(* PLC project lng-production, Generated TextualNotationConverter 1.0 *)
(* stored: creationDateTime 2025-07-30T12:00:00, modificationDateTime 2025-09-16T14:04:18 *)

FUNCTION_BLOCK ANALOG_IN
  VAR_INPUT
    Name : STRING;
    Description : STRING;
    Raw_Signal : REAL;
    PV_High : REAL;
    PV_Low : REAL;
    Scaling_Slope : REAL;
    Scaling_Offset : REAL;
    Alarm_Enable : BOOL;
  END_VAR
  VAR_OUTPUT
    PV : REAL;
    High_Alarm : BOOL;
    Low_Alarm : BOOL;
    General_Fault : BOOL;
  END_VAR

            
          
END_FUNCTION_BLOCK

FUNCTION_BLOCK RATIO_CONTROL
  VAR_INPUT
    Name : STRING;
    Description : STRING;
    Auto : BOOL;
    PrimaryPV : REAL;
    SecondaryPV : REAL;
    RatioSP : REAL;
    Bias : REAL;
    TrimKp : REAL;
    TrimTi : STRING;
    MV_MIN : REAL;
    MV_MAX : REAL;
    ManOut : REAL;
    Inhibit : BOOL;
  END_VAR
  VAR_OUTPUT
    SlaveSP : REAL;
    ActiveRatio : REAL;
    RatioErr : REAL;
  END_VAR

            
          
END_FUNCTION_BLOCK

FUNCTION_BLOCK VALVE_ELECTRIC
  VAR_INPUT
    Name : STRING;
    Description : STRING;
    Control_Signal : REAL;
    Manual_Mode : BOOL;
    Manual_Position : REAL;
    Open_Limit : REAL;
    Close_Limit : REAL;
    Timeout : STRING;
    Inhibit : BOOL;
  END_VAR
  VAR_OUTPUT
    Valve_Position : REAL;
    Feedback_Pos : REAL;
    Valve_Moving : BOOL;
    Position_Error : BOOL;
    Alarm : BOOL;
  END_VAR

            
          
END_FUNCTION_BLOCK

PROGRAM Section2
  VAR
    FT_101_Flow_PV : REAL;
    IT_102_Flow_PV : REAL;
    DP_101_DiffP_PV : REAL;
    DP_102_DiffP_PV : REAL;
    LT_101_Level_PV : REAL;
    IIC_101_LiqSepFlow_SP : REAL;
  END_VAR
  VAR
    DP-101 : ANALOG_IN;
    DP-102 : ANALOG_IN;
    FT-101 : ANALOG_IN;
    IT-102 : ANALOG_IN;
    LT-101 : ANALOG_IN;
    IIC-101 : RATIO_CONTROL;
    LCV-101 : VALVE_ELECTRIC;
  END_VAR

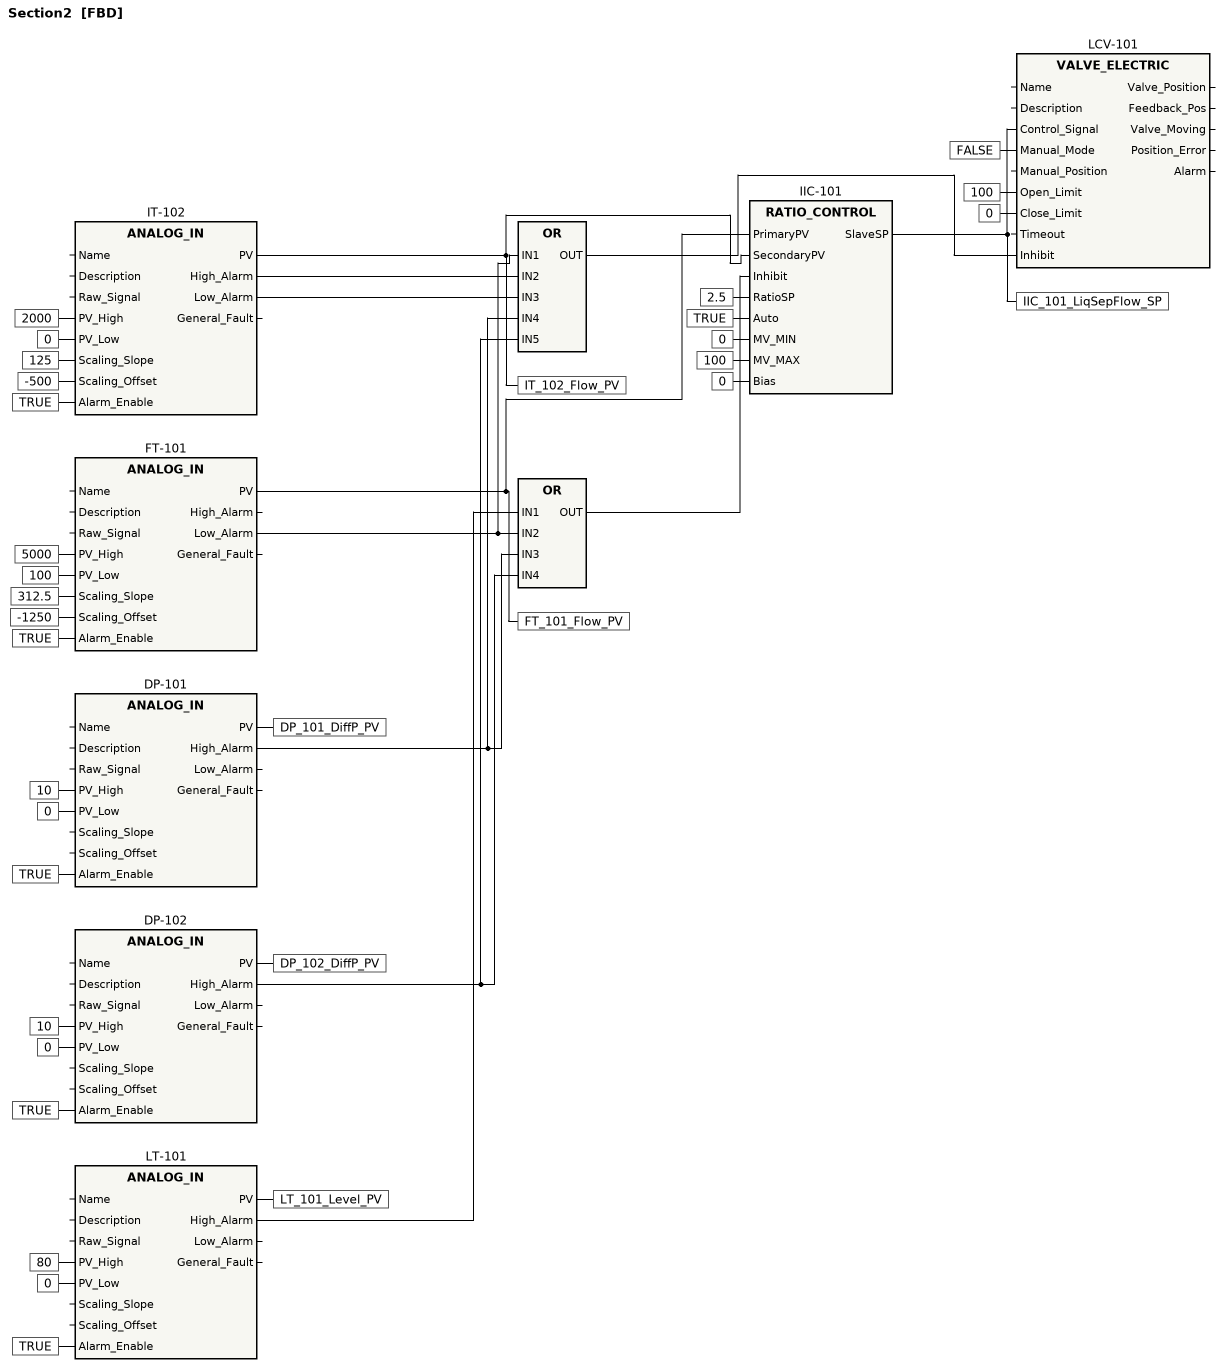
(* FBD diagram, written out as Structured Text *)
DP-101(PV_High := 10, PV_Low := 0, Alarm_Enable := TRUE);
DP_101_DiffP_PV := DP-101.PV;
DP-102(PV_High := 10, PV_Low := 0, Alarm_Enable := TRUE);
DP_102_DiffP_PV := DP-102.PV;
FT-101(PV_High := 5000, PV_Low := 100, Scaling_Slope := 312.5, Scaling_Offset := -1250, Alarm_Enable := TRUE);
FT_101_Flow_PV := FT-101.PV;
IT-102(PV_High := 2000, PV_Low := 0, Scaling_Slope := 125, Scaling_Offset := -500, Alarm_Enable := TRUE);
LT-101(PV_High := 80, PV_Low := 0, Alarm_Enable := TRUE);
IIC-101(PrimaryPV := FT-101.PV, SecondaryPV := IT-102.PV, Inhibit := LT-101.High_Alarm OR FT-101.Low_Alarm OR DP-101.High_Alarm OR DP-102.High_Alarm, RatioSP := 2.5, Auto := TRUE, MV_MIN := 0, MV_MAX := 100, Bias := 0);
IIC_101_LiqSepFlow_SP := IIC-101.SlaveSP;
IT_102_Flow_PV := IT-102.PV;
LT_101_Level_PV := LT-101.PV;
LCV-101(Control_Signal := IIC-101.SlaveSP, Manual_Mode := FALSE, Open_Limit := 100, Close_Limit := 0, Inhibit := FT-101.Low_Alarm OR IT-102.High_Alarm OR IT-102.Low_Alarm OR DP-101.High_Alarm OR DP-102.High_Alarm);
END_PROGRAM

FUNCTION_BLOCK BOOL_IN
  VAR_INPUT
    Name : STRING;
    Description : STRING;
    Bool_In : BOOL;
    Alarm_OnTrue : BOOL;
    Alarm_OnFalse : BOOL;
    Latch_Enable : BOOL;
    Reset_Latch : BOOL;
  END_VAR
  VAR_OUTPUT
    Bool_Out : BOOL;
    Alarm_Active : BOOL;
    Latched_Status : BOOL;
  END_VAR

            
          
END_FUNCTION_BLOCK

FUNCTION_BLOCK DIGITAL_IN
  VAR_INPUT
    Name : STRING;
    Description : STRING;
    DI_Raw : BOOL;
    DebounceTime : STRING;
    EnableAlarm : BOOL;
  END_VAR
  VAR_OUTPUT
    DI_Out : BOOL;
    Fault_State : BOOL;
  END_VAR

            
          
END_FUNCTION_BLOCK

FUNCTION_BLOCK DUTY_STANDBY
  VAR_INPUT
    Name : STRING;
    Description : STRING;
    Enable : BOOL;
    StartRequest : BOOL;
    AlternateEnable : BOOL;
    ForcePumpA : BOOL;
    ForcePumpB : BOOL;
    DutyElapsed : BOOL;
    MinRunElapsed : BOOL;
    SwitchoverDelayElapsed : BOOL;
    StartTimeoutElapsed : BOOL;
    PumpA_RunFB : BOOL;
    PumpB_RunFB : BOOL;
    PumpA_Fault : BOOL;
    PumpB_Fault : BOOL;
    Reset : BOOL;
    Inhibit : BOOL;
  END_VAR
  VAR_OUTPUT
    CmdPumpA : BOOL;
    CmdPumpB : BOOL;
    ActiveIsA : BOOL;
    SwitchedDueToDuty : BOOL;
    SwitchedDueToFailure : BOOL;
    Alarm_FailedStart_A : BOOL;
    Alarm_FailedStart_B : BOOL;
    Alarm_NoAvailablePump : BOOL;
  END_VAR

            
          
END_FUNCTION_BLOCK

FUNCTION_BLOCK MOTOR_2SPD
  VAR_INPUT
    Name : STRING;
    Description : STRING;
    Start_Cmd : BOOL;
    Stop_Cmd : BOOL;
    Speed_High_Cmd : BOOL;
    Speed_Low_Cmd : BOOL;
    Inhibit : BOOL;
  END_VAR
  VAR_OUTPUT
    Motor_Start_Out : BOOL;
    FB_Running : BOOL;
    FB_Trip : BOOL;
    FB_HighSpeed : BOOL;
    FB_LowSpeed : BOOL;
    Alarm_Speed_Error : BOOL;
  END_VAR

            
          
END_FUNCTION_BLOCK

FUNCTION_BLOCK MOTOR_ON_OFF
  VAR_INPUT
    Name : STRING;
    Description : STRING;
    Start_Cmd : BOOL;
    Stop_Cmd : BOOL;
    Start_Delay : STRING;
    MinRunTime : STRING;
    Inhibit : BOOL;
  END_VAR
  VAR_OUTPUT
    Motor_Start_Out : BOOL;
    FB_Running : BOOL;
    FB_Trip : BOOL;
    Alarm_Start_Fail : BOOL;
    Alarm_Stop_Fail : BOOL;
  END_VAR

            
          
END_FUNCTION_BLOCK

FUNCTION_BLOCK MOTOR_VSD
  VAR_INPUT
    Name : STRING;
    Description : STRING;
    Start_Cmd : BOOL;
    Stop_Cmd : BOOL;
    Speed_SP : REAL;
    Accel_Ramp : STRING;
    Decel_Ramp : STRING;
    Inhibit : BOOL;
  END_VAR
  VAR_OUTPUT
    Speed_Out : REAL;
    FB_Running : BOOL;
    FB_Fault : BOOL;
    FB_Ready : BOOL;
    FB_ActualSpeed : REAL;
    Alarm_Speed_Deviation : BOOL;
    Alarm_Comm_Fail : BOOL;
  END_VAR

            
          
END_FUNCTION_BLOCK

FUNCTION_BLOCK PID_BASIC
  VAR_INPUT
    Name : STRING;
    Description : STRING;
    AUTO : BOOL;
    PV : REAL;
    SP : REAL;
    MV_MIN : REAL;
    MV_MAX : REAL;
    X0 : REAL;
    KP : REAL;
    TR : REAL;
    TD : REAL;
    PV_High : REAL;
    PV_Low : REAL;
    Deviation_Limit : REAL;
    Inhibit : BOOL;
  END_VAR
  VAR_OUTPUT
    PV_High_Alarm : BOOL;
    PV_Low_Alarm : BOOL;
    Deviation_Alarm : BOOL;
    XOUT : REAL;
  END_VAR

            
          
END_FUNCTION_BLOCK

FUNCTION_BLOCK SPLIT_RANGE
  VAR_INPUT
    Name : STRING;
    Description : STRING;
    IN : REAL;
    Split_Point : REAL;
    Output1_Start : REAL;
    Output1_End : REAL;
    Output2_Start : REAL;
    Output2_End : REAL;
  END_VAR
  VAR_OUTPUT
    OUT1 : REAL;
    OUT2 : REAL;
  END_VAR

            
          
END_FUNCTION_BLOCK

FUNCTION_BLOCK VALVE_ON_OFF
  VAR_INPUT
    Name : STRING;
    Description : STRING;
    Open_Cmd : BOOL;
    Close_Cmd : BOOL;
    Timeout : STRING;
    Inhibit : BOOL;
  END_VAR
  VAR_OUTPUT
    FB_Opened : BOOL;
    FB_Closed : BOOL;
    Valve_Open_Out : BOOL;
    Valve_Close_Out : BOOL;
    Alarm_Position_Error : BOOL;
    Alarm_General : BOOL;
  END_VAR

            
          
END_FUNCTION_BLOCK

FUNCTION_BLOCK VOTING_ANALOG
  VAR_INPUT
    Name : STRING;
    Description : STRING;
    Input1 : REAL;
    Input2 : REAL;
    Input3 : REAL;
    Deviation_Limit : REAL;
    Voting_Scheme : STRING;
    EnableAlarm : BOOL;
    Inhibit : BOOL;
  END_VAR
  VAR_OUTPUT
    Voted_Output : REAL;
    Sensor1_Fault : BOOL;
    Sensor2_Fault : BOOL;
    Sensor3_Fault : BOOL;
    Alarm_Voting_Error : BOOL;
    Healthy_Sensors_Count : INT;
  END_VAR

            
          
END_FUNCTION_BLOCK

PROGRAM Section3
  VAR
    TT201_Temperature_PV : REAL;
    PT201_FlashTankPressure_PV : REAL;
    LT201_AbsorberLevel_PV : REAL;
    AI201_CO2_PV : REAL;
    TIC201_MV_SteamValveCmd : REAL;
  END_VAR
  VAR
    AI-201 : ANALOG_IN;
    LT-201 : ANALOG_IN;
    PT-201 : ANALOG_IN;
    TT-201 : ANALOG_IN;
    TIC-201 : PID_BASIC;
    FV-101 : VALVE_ELECTRIC;
  END_VAR
  VAR  (* added by the conversion: wires and edge detectors of the diagram *)
    _OR43_OUT : BOOL;
  END_VAR

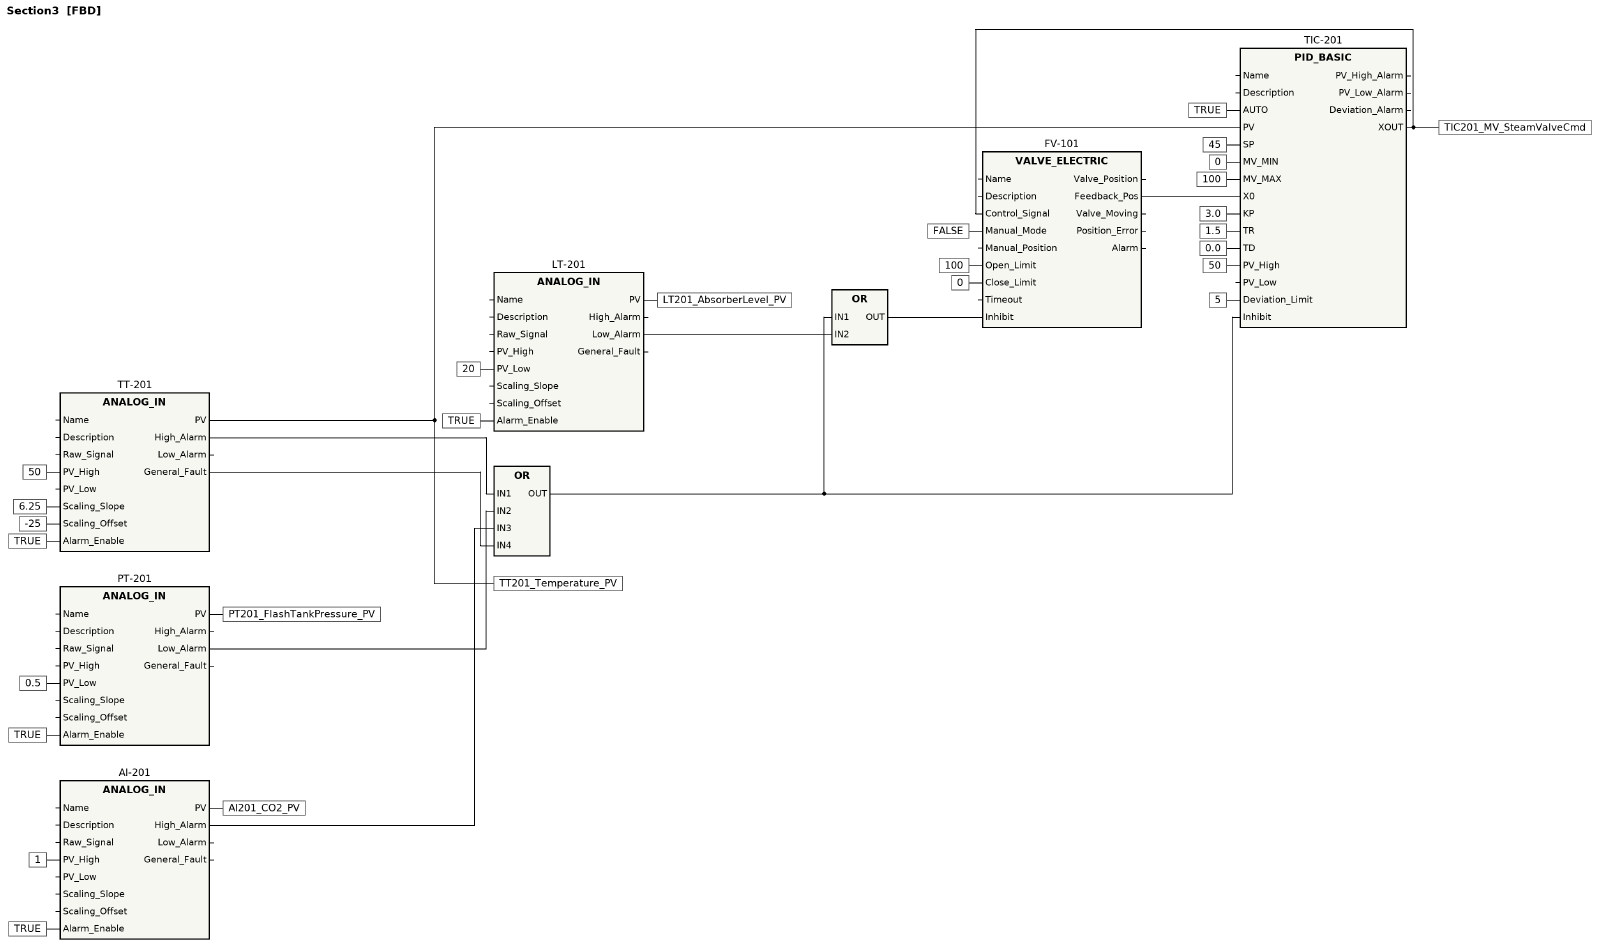
(* FBD diagram, written out as Structured Text *)
AI-201(PV_High := 1, Alarm_Enable := TRUE);
AI201_CO2_PV := AI-201.PV;
LT-201(PV_Low := 20, Alarm_Enable := TRUE);
LT201_AbsorberLevel_PV := LT-201.PV;
PT-201(PV_Low := 0.5, Alarm_Enable := TRUE);
PT201_FlashTankPressure_PV := PT-201.PV;
TT-201(PV_High := 50, Scaling_Slope := 6.25, Scaling_Offset := -25, Alarm_Enable := TRUE);
_OR43_OUT := TT-201.High_Alarm OR PT-201.Low_Alarm OR AI-201.High_Alarm OR TT-201.General_Fault;
FV-101(Control_Signal := TIC-201.XOUT, Manual_Mode := FALSE, Open_Limit := 100, Close_Limit := 0, Inhibit := _OR43_OUT OR LT-201.Low_Alarm);
TIC-201(AUTO := TRUE, PV := TT-201.PV, SP := 45, MV_MIN := 0, MV_MAX := 100, X0 := FV-101.Feedback_Pos, KP := 3.0, TR := 1.5, TD := 0.0, PV_High := 50, Deviation_Limit := 5, Inhibit := _OR43_OUT);
TIC201_MV_SteamValveCmd := TIC-201.XOUT;
TT201_Temperature_PV := TT-201.PV;
END_PROGRAM

PROGRAM Section4
  VAR
    AI302_H2O_Outlet_PV : REAL;
    AI303_Hg_Permissive_PV : REAL;
    AI304_H2O_RatioOpt_PV : REAL;
    FT301_FeedGasFlow_PV : REAL;
    DP301_MolSieveBed_DP_PV : REAL;
    FFIC303_RegenFlow_SP_to_FIC302 : REAL;
  END_VAR
  VAR
    AI-302 : ANALOG_IN;
    AI-303 : ANALOG_IN;
    AI-304 : ANALOG_IN;
    DI-301 : DIGITAL_IN;
    DP-301 : ANALOG_IN;
    FIC-302 : PID_BASIC;
    FT-301 : ANALOG_IN;
    FV-302 : VALVE_ELECTRIC;
    FFIC-303 : RATIO_CONTROL;
  END_VAR
  VAR  (* added by the conversion: wires and edge detectors of the diagram *)
    _OR78_OUT : BOOL;
  END_VAR

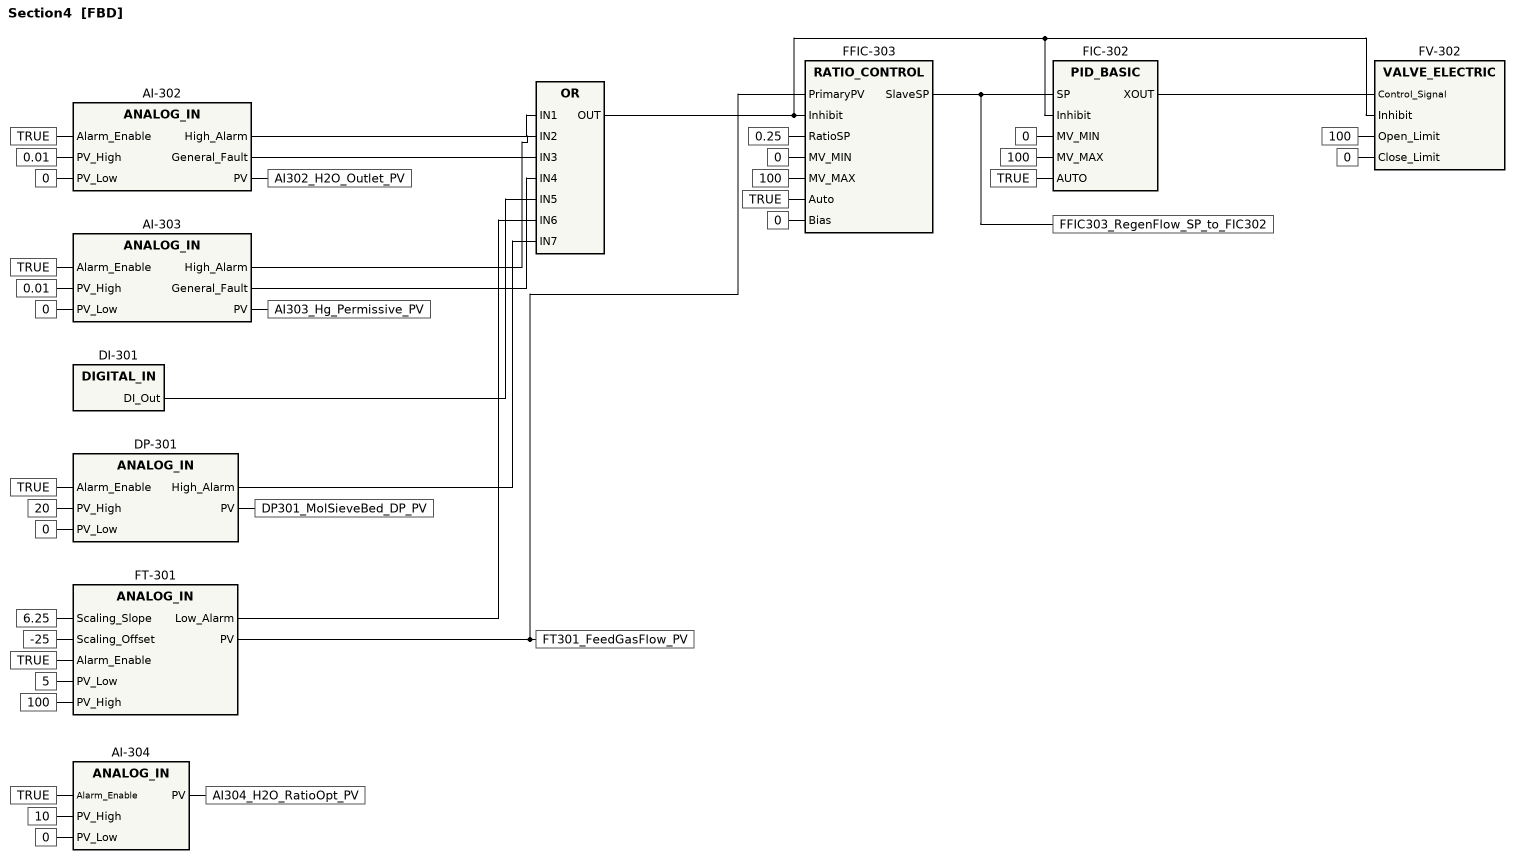
(* FBD diagram, written out as Structured Text *)
AI-302(Alarm_Enable := TRUE, PV_High := 0.01, PV_Low := 0);
AI302_H2O_Outlet_PV := AI-302.PV;
AI-303(Alarm_Enable := TRUE, PV_High := 0.01, PV_Low := 0);
AI303_Hg_Permissive_PV := AI-303.PV;
AI-304(Alarm_Enable := TRUE, PV_High := 10, PV_Low := 0);
AI304_H2O_RatioOpt_PV := AI-304.PV;
DP-301(Alarm_Enable := TRUE, PV_High := 20, PV_Low := 0);
DP301_MolSieveBed_DP_PV := DP-301.PV;
FT-301(Scaling_Slope := 6.25, Scaling_Offset := -25, Alarm_Enable := TRUE, PV_Low := 5, PV_High := 100);
DI-301();
_OR78_OUT := AI-302.High_Alarm OR AI-303.High_Alarm OR AI-302.General_Fault OR AI-303.General_Fault OR DI-301.DI_Out OR FT-301.Low_Alarm OR DP-301.High_Alarm;
FFIC-303(PrimaryPV := FT-301.PV, Inhibit := _OR78_OUT, RatioSP := 0.25, MV_MIN := 0, MV_MAX := 100, Auto := TRUE, Bias := 0);
FFIC303_RegenFlow_SP_to_FIC302 := FFIC-303.SlaveSP;
FT301_FeedGasFlow_PV := FT-301.PV;
FIC-302(SP := FFIC-303.SlaveSP, Inhibit := _OR78_OUT, MV_MIN := 0, MV_MAX := 100, AUTO := TRUE);
FV-302(Control_Signal := FIC-302.XOUT, Inhibit := _OR78_OUT, Open_Limit := 100, Close_Limit := 0);
END_PROGRAM

PROGRAM Section5
  VAR
    PVT_401_Voted_Pressure : REAL;
    TVT_402_Voted_Temperature : REAL;
  END_VAR
  VAR
    PT-401A : ANALOG_IN;
    PT-401B : ANALOG_IN;
    PT-401C : ANALOG_IN;
    TT-105 : ANALOG_IN;
    TT-106 : ANALOG_IN;
    TT-107 : ANALOG_IN;
    PVT-401 : VOTING_ANALOG;
    TVT-402 : VOTING_ANALOG;
    PIC-401 : PID_BASIC;
    TIC-402 : PID_BASIC;
    PV-102 : VALVE_ELECTRIC;
    FV-107 : VALVE_ELECTRIC;
    XV-104 : VALVE_ON_OFF;
    I-401 : BOOL_IN;
    I-402 : BOOL_IN;
    MA-401 : BOOL_IN;
  END_VAR
  VAR  (* added by the conversion: wires and edge detectors of the diagram *)
    _OR121_OUT : BOOL;
    _AND122_OUT : BOOL;
    _OR123_OUT : BOOL;
  END_VAR

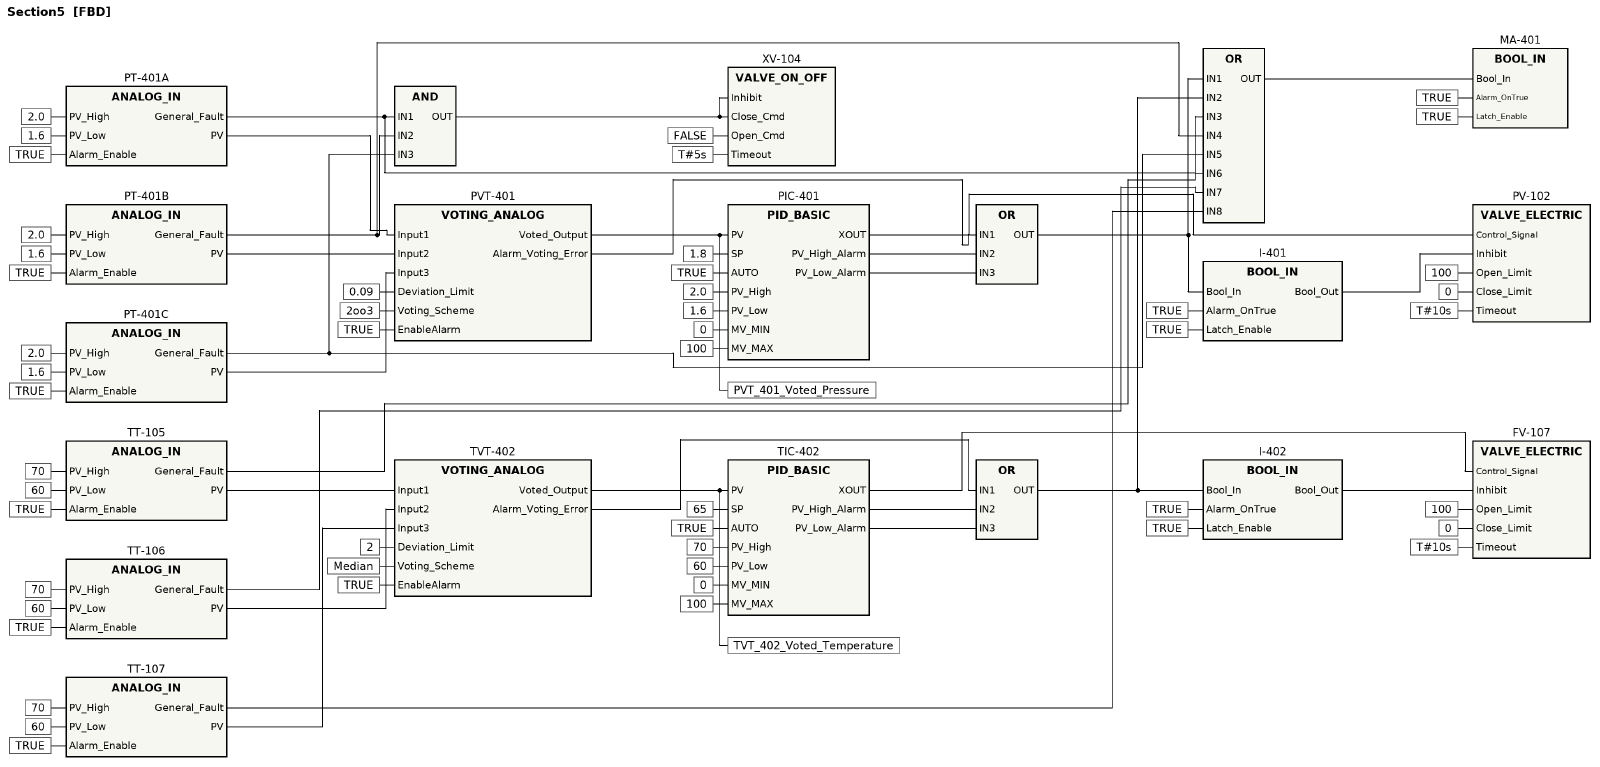
(* FBD diagram, written out as Structured Text *)
PT-401A(PV_High := 2.0, PV_Low := 1.6, Alarm_Enable := TRUE);
PT-401B(PV_High := 2.0, PV_Low := 1.6, Alarm_Enable := TRUE);
PT-401C(PV_High := 2.0, PV_Low := 1.6, Alarm_Enable := TRUE);
PVT-401(Input1 := PT-401A.PV, Input2 := PT-401B.PV, Input3 := PT-401C.PV, Deviation_Limit := 0.09, Voting_Scheme := 2oo3, EnableAlarm := TRUE);
PVT_401_Voted_Pressure := PVT-401.Voted_Output;
TT-105(PV_High := 70, PV_Low := 60, Alarm_Enable := TRUE);
TT-106(PV_High := 70, PV_Low := 60, Alarm_Enable := TRUE);
TT-107(PV_High := 70, PV_Low := 60, Alarm_Enable := TRUE);
TVT-402(Input1 := TT-105.PV, Input2 := TT-106.PV, Input3 := TT-107.PV, Deviation_Limit := 2, Voting_Scheme := Median, EnableAlarm := TRUE);
TVT_402_Voted_Temperature := TVT-402.Voted_Output;
PIC-401(PV := PVT-401.Voted_Output, SP := 1.8, AUTO := TRUE, PV_High := 2.0, PV_Low := 1.6, MV_MIN := 0, MV_MAX := 100);
_OR121_OUT := PVT-401.Alarm_Voting_Error OR PIC-401.PV_High_Alarm OR PIC-401.PV_Low_Alarm;
_AND122_OUT := PT-401A.General_Fault AND PT-401B.General_Fault AND PT-401C.General_Fault;
TIC-402(PV := TVT-402.Voted_Output, SP := 65, AUTO := TRUE, PV_High := 70, PV_Low := 60, MV_MIN := 0, MV_MAX := 100);
_OR123_OUT := TVT-402.Alarm_Voting_Error OR TIC-402.PV_High_Alarm OR TIC-402.PV_Low_Alarm;
I-401(Bool_In := _OR121_OUT, Alarm_OnTrue := TRUE, Latch_Enable := TRUE);
PV-102(Control_Signal := PIC-401.XOUT, Inhibit := I-401.Bool_Out, Open_Limit := 100, Close_Limit := 0, Timeout := T#10s);
I-402(Bool_In := _OR123_OUT, Alarm_OnTrue := TRUE, Latch_Enable := TRUE);
FV-107(Control_Signal := TIC-402.XOUT, Inhibit := I-402.Bool_Out, Open_Limit := 100, Close_Limit := 0, Timeout := T#10s);
XV-104(Inhibit := _AND122_OUT, Close_Cmd := _AND122_OUT, Open_Cmd := FALSE, Timeout := T#5s);
MA-401(Bool_In := _OR121_OUT OR _OR123_OUT OR PT-401A.General_Fault OR PT-401B.General_Fault OR PT-401C.General_Fault OR TT-105.General_Fault OR TT-106.General_Fault OR TT-107.General_Fault, Alarm_OnTrue := TRUE, Latch_Enable := TRUE);
END_PROGRAM

PROGRAM Section6
  VAR
    FT501_PropaneFlow_PV : REAL;
    FT502_MRFlow_PV : REAL;
    PT501_EndFlashDrumPressure_PV : REAL;
    TIT102_MCHE_OutletTemp_PV : REAL;
    FIC504_MRFlow_SP_From_FFIC503 : REAL;
    FFIC503_ActiveRatio : REAL;
    Operator_RatioBias : REAL;
    FFIC503_DV_HI : BOOL;
    FFIC503_DV_LO : BOOL;
  END_VAR
  VAR
    FFIC-503 : RATIO_CONTROL;
    FIC-504 : PID_BASIC;
    FV-502 : VALVE_ELECTRIC;
    FV-501 : VALVE_ELECTRIC;
    FT-501 : ANALOG_IN;
    FT-502 : ANALOG_IN;
    PT-501 : ANALOG_IN;
    TIT-102 : ANALOG_IN;
  END_VAR
  VAR  (* added by the conversion: wires and edge detectors of the diagram *)
    _TON201_OUT : BOOL;
    _OR210_OUT : BOOL;
    _OR204_OUT : BOOL;
    _OR211_OUT : BOOL;
  END_VAR

(* FBD diagram, written out as Structured Text *)
FT-501(Scaling_Slope := 312.5, Scaling_Offset := -1250.0, PV_Low := 500.0, PV_High := 5000.0, Alarm_Enable := TRUE);
FT-502(Scaling_Slope := 125.0, Scaling_Offset := -500.0, PV_Low := 200.0, PV_High := 2000.0, Alarm_Enable := TRUE);
TIT-102(PV_High := -155.0, Alarm_Enable := TRUE);
FV-501(Open_Limit := 100.0);
_TON201_OUT := TON(FV-501.Feedback_Pos > 99.0, T#5s);
PT-501(PV_Low := 2.0, Alarm_Enable := TRUE);
_OR210_OUT := FT-501.General_Fault OR FT-502.General_Fault;
_OR204_OUT := FT-501.Low_Alarm OR FT-501.High_Alarm OR FT-502.Low_Alarm OR FT-502.High_Alarm OR _OR210_OUT;
_OR211_OUT := PT-501.Low_Alarm OR _OR204_OUT;
FFIC-503(PrimaryPV := FT-501.PV, SecondaryPV := FT-502.PV, RatioSP := LIMIT(SEL(TIT-102.PV > (-155.0), 0.0, 0.1) + 2.5 + Operator_RatioBias, 2.0, 3.0), Auto := NOT (FT-501.PV < 500.0 OR _TON201_OUT OR _OR211_OUT), ManOut := SEL(SEL(_TON201_OUT, 100.0, 1000.0), _OR204_OUT, 500.0), Inhibit := _OR211_OUT);
FFIC503_ActiveRatio := FFIC-503.ActiveRatio;
FFIC503_DV_HI := TON(FFIC-503.RatioErr > 0.2, T#10s);
FFIC503_DV_LO := TON(FFIC-503.RatioErr < (-0.2), T#10s);
FIC504_MRFlow_SP_From_FFIC503 := FFIC-503.SlaveSP;
FT501_PropaneFlow_PV := FT-501.PV;
FT502_MRFlow_PV := FT-502.PV;
PT501_EndFlashDrumPressure_PV := PT-501.PV;
TIT102_MCHE_OutletTemp_PV := TIT-102.PV;
FIC-504(SP := FFIC-503.SlaveSP, PV := FT-502.PV, Inhibit := _OR210_OUT);
FV-502(Control_Signal := FIC-504.XOUT);
END_PROGRAM

PROGRAM Section7
  VAR
    FT601A_Raw_mA : REAL;
    FT601B_Raw_mA : REAL;
    LIT601_Raw_mA : REAL;
    LT601_Raw_mA : REAL;
    HS601_HandSwitch_IN : BOOL;
    FT601A_LNG_Flow_PV : REAL;
    FT601B_BOG_Flow_PV : REAL;
    FT601B_BOG_Flow_SP : REAL;
    LIT601_TankLevel_PV : REAL;
    LT601_TankLevel_PV : REAL;
  END_VAR
  VAR
    FT-601A : ANALOG_IN;
    FT-601B : ANALOG_IN;
    LIT-601 : ANALOG_IN;
    LT-601 : ANALOG_IN;
    HS-601 : BOOL_IN;
    FFIC-601 : RATIO_CONTROL;
    FIC-601B : PID_BASIC;
    FV-601B : VALVE_ELECTRIC;
    C-601 : MOTOR_ON_OFF;
  END_VAR

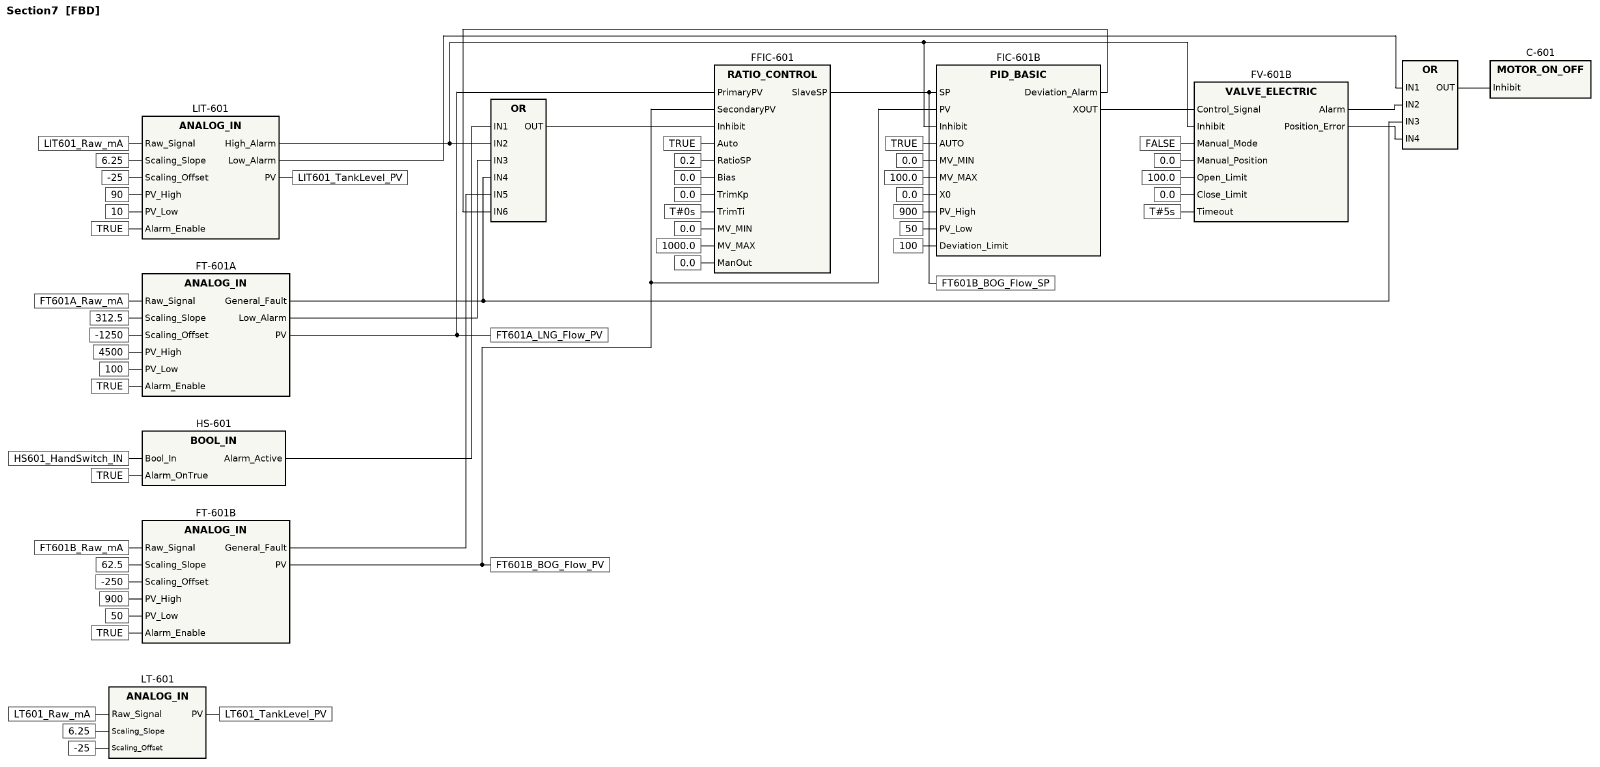
(* FBD diagram, written out as Structured Text *)
FT-601A(Raw_Signal := FT601A_Raw_mA, Scaling_Slope := 312.5, Scaling_Offset := -1250, PV_High := 4500, PV_Low := 100, Alarm_Enable := TRUE);
FT601A_LNG_Flow_PV := FT-601A.PV;
FT-601B(Raw_Signal := FT601B_Raw_mA, Scaling_Slope := 62.5, Scaling_Offset := -250, PV_High := 900, PV_Low := 50, Alarm_Enable := TRUE);
FT601B_BOG_Flow_PV := FT-601B.PV;
HS-601(Bool_In := HS601_HandSwitch_IN, Alarm_OnTrue := TRUE);
LIT-601(Raw_Signal := LIT601_Raw_mA, Scaling_Slope := 6.25, Scaling_Offset := -25, PV_High := 90, PV_Low := 10, Alarm_Enable := TRUE);
FIC-601B(SP := FFIC-601.SlaveSP, PV := FT-601B.PV, Inhibit := LIT-601.High_Alarm, AUTO := TRUE, MV_MIN := 0.0, MV_MAX := 100.0, X0 := 0.0, PV_High := 900, PV_Low := 50, Deviation_Limit := 100);
FFIC-601(PrimaryPV := FT-601A.PV, SecondaryPV := FT-601B.PV, Inhibit := HS-601.Alarm_Active OR LIT-601.High_Alarm OR FT-601A.Low_Alarm OR FT-601A.General_Fault OR FT-601B.General_Fault OR FIC-601B.Deviation_Alarm, Auto := TRUE, RatioSP := 0.2, Bias := 0.0, TrimKp := 0.0, TrimTi := T#0s, MV_MIN := 0.0, MV_MAX := 1000.0, ManOut := 0.0);
FT601B_BOG_Flow_SP := FFIC-601.SlaveSP;
LIT601_TankLevel_PV := LIT-601.PV;
LT-601(Raw_Signal := LT601_Raw_mA, Scaling_Slope := 6.25, Scaling_Offset := -25);
LT601_TankLevel_PV := LT-601.PV;
FV-601B(Control_Signal := FIC-601B.XOUT, Inhibit := LIT-601.High_Alarm, Manual_Mode := FALSE, Manual_Position := 0.0, Open_Limit := 100.0, Close_Limit := 0.0, Timeout := T#5s);
C-601(Inhibit := LIT-601.Low_Alarm OR FV-601B.Alarm OR FT-601A.General_Fault OR FV-601B.Position_Error);
END_PROGRAM

CONFIGURATION Config0
  RESOURCE Res0 ON PLC
    TASK task0(INTERVAL := T#20ms, PRIORITY := 0);
    PROGRAM instance0 WITH task0 : Section2;
    PROGRAM instance_1 WITH task0 : Section3;
    PROGRAM instance_2 WITH task0 : Section4;
    PROGRAM instance_3 WITH task0 : Section5;
    PROGRAM instance_4 WITH task0 : Section6;
    PROGRAM instance_5 WITH task0 : Section7;
  END_RESOURCE
END_CONFIGURATION
